// TIA Portal project "Distributore_bibite" (V15.1)

(* hardware
DEVICE "S7-1200 station_1"  S7-1200 Station
   slot 0: "Telaio di montaggio_0"  S7-1200 Rack  Rack  V1.0
   slot 1: "PLC_1"  CPU 1214C DC/DC/DC  6ES7 214-1AG40-0XB0  V4.2
*)

// ===== PLC "PLC_1"  CPU 1214C DC/DC/DC =====

VAR_GLOBAL   // PLC tag table "Tabella delle variabili standard"
   "moneta" AT %I0.0 : Bool;
   "fineCorsaA" AT %I0.1 : Bool;
   "fineCorsaB" AT %I0.2 : Bool;
   "bibitaPresa" AT %I0.3 : Bool;
   "SA" AT %Q0.0 : Bool;
   "SB" AT %Q0.1 : Bool;
   "blocca" AT %Q0.2 : Bool;
   "prelievo" AT %M0.0 : Bool;
END_VAR

VAR_GLOBAL CONSTANT   // PLC tag table "Tabella delle variabili standard"
   "tempo" : Time := T#5s;
END_VAR

DATA_BLOCK "variabili_stato"   // DB1
{ S7_Optimized_Access := 'TRUE' }
VERSION : 0.1
   VAR RETAIN
      home : Bool := true;
      consegnaBibita : Bool;
      rientroSB : Bool;
      NuovaBibita : Bool;
      rientroSA : Bool;
      Attesa : Bool;
   END_VAR
BEGIN
END_DATA_BLOCK

// folder: System blocks/Program resources

DATA_BLOCK "IEC_Timer_0_DB"   // DB2
{ S7_Optimized_Access := 'TRUE' }
AUTHOR : Simatic
FAMILY : IEC
NAME : IEC_TMR
VERSION : 1.0
// stored: InstanceOfName IEC_TIMER
"IEC_TIMER"
BEGIN
END_DATA_BLOCK

DATA_BLOCK "IEC_Timer_0_DB_1"   // DB3
{ S7_Optimized_Access := 'TRUE' }
AUTHOR : Simatic
FAMILY : IEC
NAME : IEC_TMR
VERSION : 1.0
// stored: InstanceOfName IEC_TIMER
"IEC_TIMER"
BEGIN
END_DATA_BLOCK

// folder: (top level)

ORGANIZATION_BLOCK "Main"   // OB1, LAD, ProgramCycle
TITLE = "Main Program Sweep (Cycle)"
{ S7_Optimized_Access := 'TRUE' }
VERSION : 0.1
   VAR_INPUT
      Initial_Call : Bool;   // Initial call of this OB
      Remanence : Bool;   // =True, if remanent data are available
   END_VAR
BEGIN

REGION Network 1
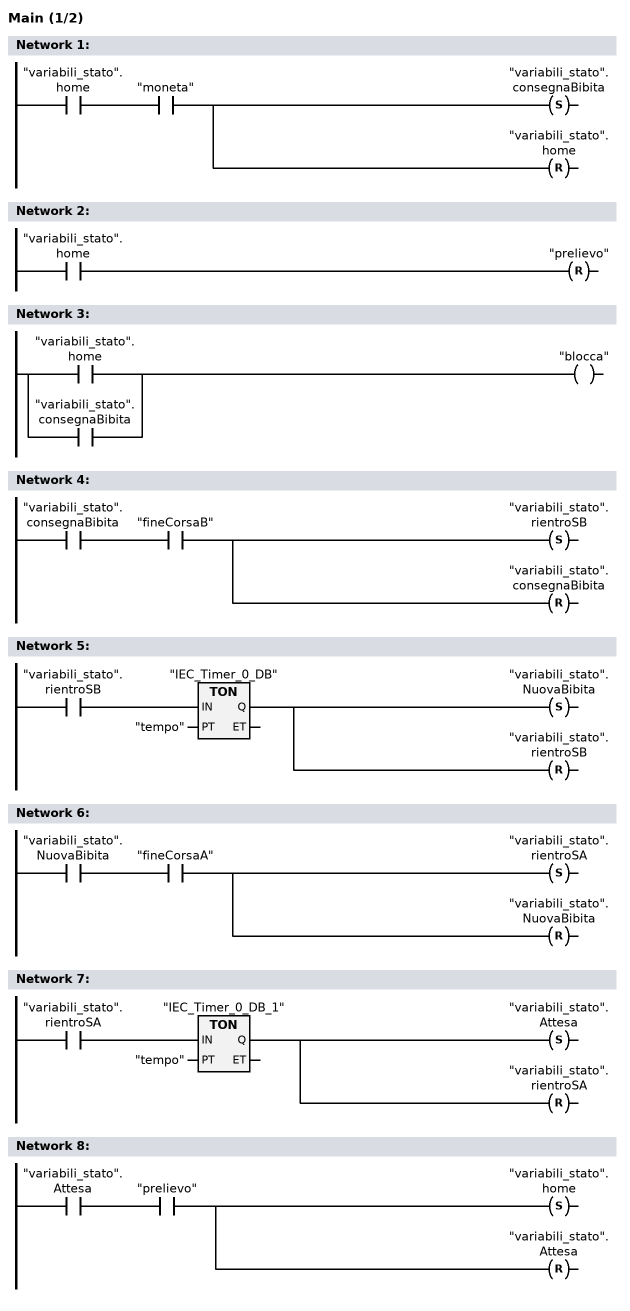
   RUNG wire#powerrail
      Contact( "variabili_stato".home )
      Contact( "moneta" )
      wire#w1
      S_Coil( "variabili_stato".consegnaBibita )
   END_RUNG
   RUNG wire#w1
      R_Coil( "variabili_stato".home )
   END_RUNG
   // the same network as SCL:
   IF "variabili_stato".home AND "moneta" THEN
       "variabili_stato".consegnaBibita := TRUE;
       "variabili_stato".home := FALSE;
   END_IF;
END_REGION

REGION Network 2
   RUNG wire#powerrail
      Contact( "variabili_stato".home )
      R_Coil( "prelievo" )
   END_RUNG
   // the same network as SCL:
   IF "variabili_stato".home THEN "prelievo" := FALSE; END_IF;
END_REGION

REGION Network 3
   RUNG wire#powerrail
      Contact( "variabili_stato".home )
      wire#w1
      Coil( "blocca" )
   END_RUNG
   RUNG wire#powerrail
      Contact( "variabili_stato".consegnaBibita )
   END_RUNG wire#w1
   // the same network as SCL:
   "blocca" := "variabili_stato".home OR "variabili_stato".consegnaBibita;
END_REGION

REGION Network 4
   RUNG wire#powerrail
      Contact( "variabili_stato".consegnaBibita )
      Contact( "fineCorsaB" )
      wire#w1
      S_Coil( "variabili_stato".rientroSB )
   END_RUNG
   RUNG wire#w1
      R_Coil( "variabili_stato".consegnaBibita )
   END_RUNG
   // the same network as SCL:
   IF "variabili_stato".consegnaBibita AND "fineCorsaB" THEN
       "variabili_stato".rientroSB := TRUE;
       "variabili_stato".consegnaBibita := FALSE;
   END_IF;
END_REGION

REGION Network 5
   "IEC_Timer_0_DB".TON(IN := "variabili_stato".rientroSB, PT := "tempo");
   IF "IEC_Timer_0_DB".Q THEN
       "variabili_stato".NuovaBibita := TRUE;
       "variabili_stato".rientroSB := FALSE;
   END_IF;
END_REGION

REGION Network 6
   RUNG wire#powerrail
      Contact( "variabili_stato".NuovaBibita )
      Contact( "fineCorsaA" )
      wire#w1
      S_Coil( "variabili_stato".rientroSA )
   END_RUNG
   RUNG wire#w1
      R_Coil( "variabili_stato".NuovaBibita )
   END_RUNG
   // the same network as SCL:
   IF "variabili_stato".NuovaBibita AND "fineCorsaA" THEN
       "variabili_stato".rientroSA := TRUE;
       "variabili_stato".NuovaBibita := FALSE;
   END_IF;
END_REGION

REGION Network 7
   "IEC_Timer_0_DB_1".TON(IN := "variabili_stato".rientroSA, PT := "tempo");
   IF "IEC_Timer_0_DB_1".Q THEN
       "variabili_stato".Attesa := TRUE;
       "variabili_stato".rientroSA := FALSE;
   END_IF;
END_REGION

REGION Network 8
   RUNG wire#powerrail
      Contact( "variabili_stato".Attesa )
      Contact( "prelievo" )
      wire#w1
      S_Coil( "variabili_stato".home )
   END_RUNG
   RUNG wire#w1
      R_Coil( "variabili_stato".Attesa )
   END_RUNG
   // the same network as SCL:
   IF "variabili_stato".Attesa AND "prelievo" THEN
       "variabili_stato".home := TRUE;
       "variabili_stato".Attesa := FALSE;
   END_IF;
END_REGION

REGION Network 9
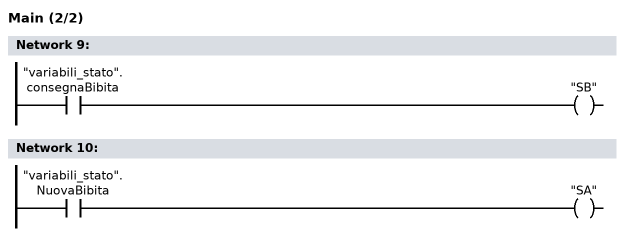
   RUNG wire#powerrail
      Contact( "variabili_stato".consegnaBibita )
      Coil( "SB" )
   END_RUNG
   // the same network as SCL:
   "SB" := "variabili_stato".consegnaBibita;
END_REGION

REGION Network 10
   RUNG wire#powerrail
      Contact( "variabili_stato".NuovaBibita )
      Coil( "SA" )
   END_RUNG
   // the same network as SCL:
   "SA" := "variabili_stato".NuovaBibita;
END_REGION
END_ORGANIZATION_BLOCK

ORGANIZATION_BLOCK "Hardware interrupt"   // OB40, LAD, HWProcessInterrupt
{ S7_Optimized_Access := 'TRUE' }
VERSION : 0.1
   VAR_INPUT
      LADDR : Hw_Io;   // Hardware identifier
      USI : Word;   // User structure identifier
      IChannel : USInt;   // Interrupt channel number
      EventType : Byte;   // EventType
   END_VAR
BEGIN

REGION Network 1
   // Il programma viene eseguito solo una volta, quindi serve un set. Un coil normale non serve a nulla.
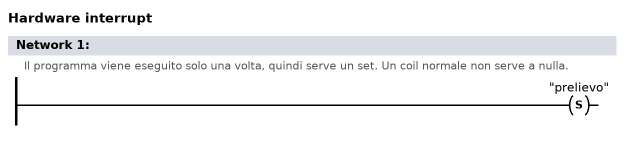
   RUNG wire#powerrail
      S_Coil( "prelievo" )
   END_RUNG
   // the same network as SCL:
   "prelievo" := TRUE;
END_REGION
END_ORGANIZATION_BLOCK